// TwinCAT 3 PLC project LabExercise
// ProgramVersion: 3.1.4023.0
// libraries:
//   Tc2_NCI, * (Beckhoff Automation GmbH)
//   Tc2_Standard, * (Beckhoff Automation GmbH)
//   Tc2_System, * (Beckhoff Automation GmbH)
//   Tc3_Module, * (Beckhoff Automation GmbH)
//   VisuDialogs, * (System)
// project tree:
//   Comissioning/Function blocks/ FB_ModifyAutomaticControlSettings.TcPOU
//   Comissioning/GVLs/ G_Commissioning.TcGVL
//   Comissioning/Struct/ ST_AutomaticControlSettings.TcDUT, ST_ClosedLoopControlSettings.TcDUT, ST_MotionReferenceGeneratorSettings.TcDUT, ST_OpenLoopControlSettings.TcDUT
//   ControlBox/Interfaces/ I_ControlBox.TcIO
//   ControlBox/Function blocks/ FB_ControlBox.TcPOU, FB_RealControlBox.TcPOU, FB_VirtualControlBox.TcPOU
//   CraneControl/Function blocks/Sub blocks/ FB_ActiveDamping.TcPOU, FB_Clock.TcPOU, FB_ClosedLoopControl.TcPOU, FB_Joystick.TcPOU, FB_MotionReferenceGenerator_limit.TcPOU, FB_OpenLoopControl.TcPOU, FB_ResetIntegralController.TcPOU, FB_Status.TcPOU
//   CraneControl/Functions/ F_BarToEng.TcPOU, F_BoomAnimation.TcPOU, F_LminToEng.TcPOU, F_PistonDisplacementToBoomAngle.TcPOU, F_RadToDeg.TcPOU
//   CraneControl/Enums/ E_Mode.TcDUT, E_Status.TcDUT
//   CraneControl/Function blocks/Main blocks/ FB_AutomaticControl.TcPOU, FB_ManualControl.TcPOU
//   CraneControl/GVLs/ G_Parameters.TcGVL, G_Work.TcGVL
//   CraneControl/Struct/ ST_ActiveDamping.TcDUT, ST_AnimationScaling.TcDUT, ST_CraneKinematics.TcDUT, ST_Parameters.TcDUT, ST_RelativeMovement.TcDUT
//   / GlobalTextList.TcGTLO, PlcTask.TcTTO, Simulator.TcTTO, Visualization Manager.TcVMO (not stored)
//   HMI/ HMI.TcVIS
//   HMI/Sub/ CommissioningHMI.TcVIS, Animation.TcVIS, VirtualControlBox.TcVIS
//   ControlBox/GVLs/ G_VirtualControlBox.TcGVL
//   Programs/ MAIN.TcPOU, P_Commissioning.TcPOU, P_ControlBox.TcPOU, P_CraneControl.TcPOU, P_Simulator.TcPOU
//   Simulator/ FB_CraneSimulator.TcPOU, G_Simulator.TcGVL
// real-time tasks:
//   TASK PlcTask: cycle T#1ms, priority 20, ADS port 350
//   TASK Simulator: cycle T#100us, priority 1, ADS port 351

CONFIGURATION LabExercise
    RESOURCE PLC ON TwinCAT3
        TASK PlcTask(INTERVAL := T#1ms, PRIORITY := 20);
        TASK Simulator(INTERVAL := T#100us, PRIORITY := 1);
        PROGRAM MAIN WITH PlcTask : MAIN;
        PROGRAM P_Simulator WITH Simulator : P_Simulator;
    END_RESOURCE
END_CONFIGURATION

// ---- Comissioning/Struct/ST_AutomaticControlSettings.TcDUT
TYPE ST_AutomaticControlSettings :
STRUCT
	bEnableVelocityFeedForwardControl	: BOOL;
	bEnableClosedLoopPositionControl	: BOOL;
	bEnableIntegralController 			: BOOL;
	bEnableActiveDamping 				: BOOL;	
END_STRUCT
END_TYPE

// ---- Comissioning/Struct/ST_ClosedLoopControlSettings.TcDUT
TYPE ST_ClosedLoopControlSettings :
STRUCT
	fMaxPositionError 					: LREAL := 1E-3;
	fProportionalGain 					: LREAL := 29.17;
	fIntegralGain 						: LREAL := 19.49;
END_STRUCT
END_TYPE

// ---- Comissioning/Struct/ST_MotionReferenceGeneratorSettings.TcDUT
TYPE ST_MotionReferenceGeneratorSettings :
STRUCT
	fStartPosition_m		: LREAL := 0.0;
	fStartVelocity_m		: LREAL	:= 0.0;
	fPositionSetpoint_ms	: LREAL := 0.25;
	fVelocitySetpoint_m		: LREAL := 0.025;
	fMaxPosition 			: LREAL := 0.45;
	fMinPosition 			: LREAL := 0.0;
	fMaxVelocity 			: LREAL := 0.05;
	fTimeBeforeStarting_s	: LREAL := 3.0;
	fRampTime_s				: LREAL := 1.0;
	fHoldPositionTime_s		: LREAL := 5.0;
END_STRUCT
END_TYPE

// ---- Comissioning/Struct/ST_OpenLoopControlSettings.TcDUT
TYPE ST_OpenLoopControlSettings :
STRUCT
	fBoreArea 			: LREAL := 0.0033183;
	fAnnulusArea 		: LREAL := 0.0023562;
	fMaxFlowCapacity 	: LREAL := 30; //[l/min]
END_STRUCT
END_TYPE

// ---- CraneControl/Enums/E_Mode.TcDUT
{attribute 'qualified_only'}
{attribute 'strict'}
TYPE E_Mode :
(
	Off,
	Manual,
	Auto
);
END_TYPE

// ---- CraneControl/Enums/E_Status.TcDUT
{attribute 'qualified_only'}
{attribute 'strict'}
TYPE E_Status :
(
	Off,
	Fault,
	Ready,
	Starting,
	Running,
	Stopping,
	Checking
);
END_TYPE

// ---- CraneControl/Struct/ST_ActiveDamping.TcDUT
TYPE ST_ActiveDamping :
STRUCT
	fFlowGainInverse : LREAL := 1.7153E03;	
	fHPF_Num1 : LREAL := 9.016E-12;
	fHPF_Num2 : LREAL := -9.016E-12;
	fHPF_Den1 : LREAL := 1.0;
	fHPF_Den2 : LREAL := -0.9905;
	fVDI_Num1 : LREAL := 25;
	fVDI_Num2 : LREAL := -48.83;
	fVDI_Num3 : LREAL := 23.85;
	fVDI_Den1 : LREAL := 1;
	fVDI_Den2 : LREAL := -1.721;
	fVDI_Den3 : LREAL := 0.7408;
END_STRUCT
END_TYPE

// ---- CraneControl/Struct/ST_AnimationScaling.TcDUT
TYPE ST_AnimationScaling :
STRUCT
	fPistonScale : LREAL := 200;
	fBoomScale : LREAL := 50;
END_STRUCT
END_TYPE

// ---- CraneControl/Struct/ST_CraneKinematics.TcDUT
TYPE ST_CraneKinematics :
STRUCT
	ABx : LREAL := 0.427;
	ABy : LREAL := 1.057;
	ACx : LREAL := 0.49484;
	ACy : LREAL := 0.133;
	fBoomLength : LREAL := 3.4;
END_STRUCT
END_TYPE

// ---- CraneControl/Struct/ST_Parameters.TcDUT
TYPE ST_Parameters :
STRUCT
	fCyclicTime 						: LREAL := 0.001; //[s]
	fMaxVelocityLimit 					: LREAL := 0.05; //[m/s]
	stOpenLoopControlSettings 			: ST_OpenLoopControlSettings;
	stClosedLoopControlSettings 		: ST_ClosedLoopControlSettings;
	stPressureFeedback 					: ST_ActiveDamping;
	stCraneKinematics 					: ST_CraneKinematics;
	stAnimationScaling 					: ST_AnimationScaling;
END_STRUCT
END_TYPE

// ---- CraneControl/Struct/ST_RelativeMovement.TcDUT
TYPE ST_RelativeMovement :
STRUCT
	pt0_x : INT := 0;
	pt0_y : INT := 0;
	pt1_x : INT := 0;
	pt1_y : INT := 0; 
END_STRUCT
END_TYPE

// ---- Comissioning/GVLs/G_Commissioning.TcGVL
{attribute 'qualified_only'}
VAR_GLOBAL
	bSetNewMaxFlowCapacity		: BOOL;
	fNewMaxFlowCapacity 		: LREAL;
	bSetNewProportionalGain 	: BOOL;
	bSetNewIntegralGain 		: BOOL;
	fNewProportionalGain 		: LREAL;
	fNewIntegralGain 			: LREAL;
	bSetNewMaxPositionError 			: BOOL;
	fNewMaxPositionError				: LREAL;
	stAutomaticControlSettings 	: ST_AutomaticControlSettings;
	stMotionReferenceGeneratorSettings  : ST_MotionReferenceGeneratorSettings;
END_VAR

// ---- CraneControl/GVLs/G_Parameters.TcGVL
{attribute 'qualified_only'}
VAR_GLOBAL
	stParam : ST_Parameters;
END_VAR

// ---- CraneControl/GVLs/G_Work.TcGVL
{attribute 'qualified_only'}
VAR_GLOBAL
	eMode 			: E_Mode;
	eStatus 		: E_Status;
	fJoystickY 		: LREAL;
	bFault 			: BOOL;
	bStartButton 	: BOOL;
	bStopButton 	: BOOL;
	fControlOutputNormalized : LREAL;
END_VAR

// ---- ControlBox/GVLs/G_VirtualControlBox.TcGVL
{attribute 'qualified_only'}
VAR_GLOBAL
	bOnSelector : BOOL;
	bAutoSelector : BOOL;
	bStartButton : BOOL;
	bStopButton : BOOL;
	fJoystickY : LREAL;
	bGreenLight : BOOL;
	bRedLight : BOOL;
END_VAR

// ---- Simulator/G_Simulator.TcGVL
{attribute 'qualified_only'}
VAR_GLOBAL
	bSimulatorOn : BOOL;
	fPistonSidePressure : LREAL;
	fRodSidePressure 	: LREAL;
	fPistonPosition 	: LREAL;
	stPistonAnimation 	: ST_RelativeMovement;
	fBoomAngle 			: LREAL;
	stBoomAnimation 	: ST_RelativeMovement;
	fBoomAnimation 		: LREAL;
	fBoomAngleDeg 		: LREAL;
END_VAR

// ---- ControlBox/Interfaces/I_ControlBox.TcIO
INTERFACE I_ControlBox

METHOD Joystick
VAR_INPUT
	eMode 	: E_Mode;
	eStatus : E_Status;
END_VAR
VAR_OUTPUT
	fJoystickY : LREAL;
END_VAR
END_METHOD

METHOD Lamps 
VAR_INPUT
	eMode 	: E_Mode;
	eStatus : E_Status;
END_VAR
END_METHOD

METHOD ModeSelector 
VAR_INPUT
END_VAR
VAR_OUTPUT
	eMode : E_Mode;
END_VAR
END_METHOD

METHOD PushButtons
VAR_INPUT
	eMode 	: E_Mode;
	eStatus : E_Status;
END_VAR
VAR_OUTPUT
	bStart : BOOL;
	bStop : BOOL;
END_VAR
END_METHOD

END_INTERFACE

// ---- Programs/MAIN.TcPOU
PROGRAM MAIN
VAR
	bActivateMotion:BOOL;		//receive from ROS    sends start and stop signal
	bAuto : BOOL;				//receive from ROS    is true if we want auto mode
	bManual : BOOL;				//receive from ROS    is true if we want manual mode
	fBoomAngleRef:LREAL;			//receive from ROS	  is the desired position for the angle of the boom
	
	fPrPist : LREAL;			//sent to ROS - pressure in piston side
	fPrRod : LREAL;				//sent to ROS - pressure in rod side
	fBoomAngle:LREAL;			//sent to ROS - is the actual boom angle while crane is moving

END_VAR

P_Commissioning();
P_ControlBox();
P_CraneControl();

//SENDING TO ROS
fPrPist := G_Simulator.fPistonSidePressure;
fPrRod := G_Simulator.fRodSidePressure;
fBoomAngle := -1 * G_Simulator.fBoomAngle;


//RECEIVING FROM ROS



	
// start or stop system (through HMI buttons)
IF bActivateMotion THEN
	G_Work.bStartButton := TRUE;   //or G_Simulator.bSimulatorOn := bActivateMotion;
//ELSE
	//G_Work.bStopButton 	:= TRUE;
END_IF 

//auto or manual selection (through HMI variables)
IF bAuto THEN
	G_VirtualControlBox.bAutoSelector := FALSE;
	// set reference position
	G_VirtualControlBox.fJoystickY	:= 1 * fBoomAngleRef;				//OROR    fBoomAnimation 		: LREAL;	OR //	fBoomAngleDeg 		: LREAL;

END_IF
	
IF bManual THEN 
	G_VirtualControlBox.bAutoSelector := FALSE;
END_IF

END_PROGRAM

// ---- Programs/P_Commissioning.TcPOU
PROGRAM P_Commissioning
VAR
	fbModifyAutomaticControlSettings : FB_ModifyAutomaticControlSettings;
END_VAR

fbModifyAutomaticControlSettings(
	stParamOpenLoopControllSettings := G_Parameters.stParam.stOpenLoopControlSettings,
	bSetNewMaxFlowCapacity := G_Commissioning.bSetNewMaxFlowCapacity,
	fNewMaxFlowCapacity := G_Commissioning.fNewMaxFlowCapacity,
	stParamClosedLoopControllSettings := G_Parameters.stParam.stClosedLoopControlSettings,	
	bSetNewProportionalGain := G_Commissioning.bSetNewProportionalGain,
	fNewProportionalGain := G_Commissioning.fNewProportionalGain,
	bSetNewIntegralGain := G_Commissioning.bSetNewIntegralGain,
	fNewIntegralGain := G_Commissioning.fNewIntegralGain,
	bSetNewMaxPositionError := G_Commissioning.bSetNewMaxPositionError,
	fNewMaxPositionError := G_Commissioning.fNewMaxPositionError
);

END_PROGRAM

// ---- Comissioning/Function blocks/FB_ModifyAutomaticControlSettings.TcPOU
FUNCTION_BLOCK FB_ModifyAutomaticControlSettings
VAR_INPUT
	stParamOpenLoopControllSettings 	: REFERENCE TO ST_OpenLoopControlSettings;
	bSetNewMaxFlowCapacity				: BOOL;
	fNewMaxFlowCapacity 				: LREAL;
	stParamClosedLoopControllSettings 	: REFERENCE TO ST_ClosedLoopControlSettings;
	bSetNewProportionalGain 			: BOOL;
	bSetNewIntegralGain 				: BOOL;
	fNewProportionalGain 				: LREAL;
	fNewIntegralGain 					: LREAL;
	bSetNewMaxPositionError 			: BOOL;
	fNewMaxPositionError				: LREAL;
END_VAR
VAR_OUTPUT
END_VAR
VAR
END_VAR

IF bSetNewMaxFlowCapacity THEN
	stParamOpenLoopControllSettings.fMaxFlowCapacity := fNewMaxFlowCapacity;
	bSetNewMaxFlowCapacity := FALSE;
END_IF

IF bSetNewProportionalGain THEN
	stParamClosedLoopControllSettings.fProportionalGain := fNewProportionalGain;
	bSetNewProportionalGain := FALSE;
END_IF

IF bSetNewIntegralGain THEN
	stParamClosedLoopControllSettings.fIntegralGain := fNewIntegralGain;
	bSetNewIntegralGain := FALSE;
END_IF

IF bSetNewMaxPositionError THEN
	stParamClosedLoopControllSettings.fMaxPositionError:= fNewMaxPositionError;
	bSetNewMaxPositionError := FALSE;
END_IF

END_FUNCTION_BLOCK

// ---- Programs/P_ControlBox.TcPOU
PROGRAM P_ControlBox
VAR
	fbControlBox : FB_ControlBox; 
END_VAR

fbControlBox(
bRealControlBox := FALSE,
eStatus := G_Work.eStatus,
eMode => G_Work.eMode,
);

END_PROGRAM

// ---- ControlBox/Function blocks/FB_ControlBox.TcPOU
FUNCTION_BLOCK FB_ControlBox
VAR_INPUT
	bRealControlBox : BOOL;
	eStatus : E_Status;
END_VAR
VAR_OUTPUT
	eMode : E_Mode;
END_VAR
VAR
	fbVirtualControlBox : FB_VirtualControlBox;
	fbRealControlBox : FB_RealControlBox;
	fbSelectedControlBox : I_ControlBox := fbVirtualControlBox;
END_VAR

IF bRealControlBox THEN
	fbSelectedControlBox := fbRealControlBox;
ELSE
	fbSelectedControlBox := fbVirtualControlBox;
END_IF	
	
fbSelectedControlBox.ModeSelector(
	eMode => eMode
);

fbSelectedControlBox.PushButtons(
	eMode := eMode,
	eStatus := eStatus,
	bStart => G_Work.bStartButton,
	bStop => G_Work.bStopButton 	
);

fbSelectedControlBox.Lamps(
	eMode := eMode,
	eStatus := eStatus
);

fbSelectedControlBox.Joystick(
	eMode := eMode,
	eStatus := eStatus,
	fJoystickY => G_Work.fJoystickY
);

//IF G_Work.eStatus = E_Status.Running THEN
//	G_VirtualControlBox.bGreenLight :=  TRUE;
//ELSE
//	G_VirtualControlBox.bGreenLight :=  FALSE;
//END_IF

//IF G_Work.eStatus = E_Status.Fault THEN
//	G_VirtualControlBox.bRedLight :=  TRUE;
//ELSE
//	G_VirtualControlBox.bRedLight :=  FALSE;
//END_IF

END_FUNCTION_BLOCK

// ---- ControlBox/Function blocks/FB_VirtualControlBox.TcPOU
FUNCTION_BLOCK FB_VirtualControlBox IMPLEMENTS I_ControlBox
VAR_INPUT
END_VAR
VAR_OUTPUT
END_VAR
VAR
END_VAR

METHOD Joystick
VAR_INPUT
	eMode 	: E_Mode;
	eStatus : E_Status;
END_VAR
VAR_OUTPUT
	fJoystickY : LREAL;
END_VAR
IF eMode = E_Mode.Manual AND eStatus = E_Status.Running THEN
	fJoystickY := G_VirtualControlBox.fJoystickY;
ELSE
	fJoystickY := 0.0;
END_IF
END_METHOD

METHOD Lamps
VAR_INPUT
	eMode 	: E_Mode;
	eStatus : E_Status;
END_VAR
IF eStatus = E_Status.Running AND NOT(eMode = E_Mode.Off) THEN
	G_VirtualControlBox.bGreenLight :=  TRUE;
ELSE
	G_VirtualControlBox.bGreenLight :=  FALSE;
END_IF

IF eStatus = E_Status.Fault  AND NOT(eMode = E_Mode.Off) THEN
	G_VirtualControlBox.bRedLight :=  TRUE;
ELSE
	G_VirtualControlBox.bRedLight :=  FALSE;
END_IF
END_METHOD

METHOD ModeSelector 
VAR_INPUT
END_VAR
VAR_OUTPUT
	eMode : E_Mode;
END_VAR
CASE eMode OF 
	E_Mode.Off:	
		IF G_VirtualControlBox.bOnSelector AND NOT(G_VirtualControlBox.bAutoSelector) THEN	
			eMode := E_Mode.Manual;
		END_IF
		
		IF G_VirtualControlBox.bOnSelector AND G_VirtualControlBox.bAutoSelector THEN	
			eMode := E_Mode.Auto;
		END_IF

	E_Mode.Manual: 
		IF NOT(G_VirtualControlBox.bOnSelector) THEN	
			eMode := E_Mode.Off;
		END_IF
		
		IF G_VirtualControlBox.bOnSelector AND G_VirtualControlBox.bAutoSelector THEN	
			eMode := E_Mode.Auto;
		END_IF
	
	E_Mode.Auto:
		IF NOT(G_VirtualControlBox.bOnSelector) THEN	
			eMode := E_Mode.Off;
		END_IF
		
		IF G_VirtualControlBox.bOnSelector AND NOT(G_VirtualControlBox.bAutoSelector) THEN	
			eMode := E_Mode.Manual;
		END_IF	
ELSE 	
	eMode := E_Mode.Off;
END_CASE
END_METHOD

METHOD PushButtons
VAR_INPUT
	eMode 	: E_Mode;
	eStatus : E_Status;
END_VAR
VAR_OUTPUT
	bStart : BOOL;
	bStop : BOOL;
END_VAR
IF NOT(eMode = E_Mode.Off) AND (NOT(eStatus = E_Status.Fault) OR (eStatus = E_Status.Off)) THEN 
	bStart := G_VirtualControlBox.bStartButton;
	bStop := G_VirtualControlBox.bStopButton;
ELSE
	bStart := FALSE;
	bStop := FALSE;
END_IF
END_METHOD

END_FUNCTION_BLOCK

// ---- ControlBox/Function blocks/FB_RealControlBox.TcPOU
FUNCTION_BLOCK FB_RealControlBox IMPLEMENTS I_ControlBox
VAR_INPUT
END_VAR
VAR_OUTPUT
END_VAR
VAR
END_VAR

METHOD Joystick
VAR_INPUT
	eMode 	: E_Mode;
	eStatus : E_Status;
END_VAR
VAR_OUTPUT
	fJoystickY : LREAL;
END_VAR
END_METHOD

METHOD Lamps 
VAR_INPUT
	eMode 	: E_Mode;
	eStatus : E_Status;
END_VAR
// To Do LAB #12
END_METHOD

METHOD ModeSelector 
VAR_INPUT
END_VAR
VAR_OUTPUT
	eMode : E_Mode;
END_VAR
// To Do LAB #12
END_METHOD

METHOD PushButtons
VAR_INPUT
	eMode 	: E_Mode;
	eStatus : E_Status;
END_VAR
VAR_OUTPUT
	bStart : BOOL;
	bStop : BOOL;
END_VAR
END_METHOD

END_FUNCTION_BLOCK

// ---- Programs/P_CraneControl.TcPOU
PROGRAM P_CraneControl
VAR
 	fbStatus 					: FB_Status;
	fbRunningClock 				: FB_Clock;
	fbManualControl 			: FB_ManualControl; 
	bEnableManualControl 		: BOOL;
	fbAutomaticControl 			: FB_AutomaticControl;
	bEnableAutomaticControl 	: BOOL; 
	fbActiveDamping 			: FB_ActiveDamping;
	fControlOutputNormalized 	: LREAL; 
END_VAR

fbStatus(
bFault := G_Work.bFault,
eMode := G_Work.eMode,
fTime := fbRunningClock.fTime,
eStatus => G_Work.eStatus
);

fbRunningClock(
	bStart := (fbStatus.eStatus = E_Status.Starting) OR (fbStatus.eStatus = E_Status.Running),
	bStop := (fbStatus.eStatus = E_Status.Stopping),
	fCycleTime := G_Parameters.stParam.fCyclicTime
);

fbManualControl(
	eMode := G_Work.eMode,
	eStatus := G_Work.eStatus,
	stParam := G_Parameters.stParam, 
);

fbAutomaticControl(
	eMode := G_Work.eMode,
	eStatus := G_Work.eStatus,
	stAutomaticControlSettings := G_Commissioning.stAutomaticControlSettings,
	stMotionReferenceGeneratorSettings := G_Commissioning.stMotionReferenceGeneratorSettings,
	stParam := G_Parameters.stParam,
	fPositionFeedback := G_Simulator.fPistonPosition
);

fbActiveDamping(
	ssMethodType := BOOL_TO_SINT(G_Commissioning.stAutomaticControlSettings.bEnableActiveDamping),
	bEnable := (fbStatus.eStatus = E_Status.Running),
	stParam := G_Parameters.stParam,
	fPressurePistonSide_Pa := G_Simulator.fPistonSidePressure,
	fPressureRodSide_Pa := G_Simulator.fRodSidePressure
);
 
IF (G_Work.eMode = E_Mode.Manual AND G_Work.eStatus = E_Status.Running) THEN
	fControlOutputNormalized := LIMIT(-1.0, (fbManualControl.fControlOutputNormalized - fbActiveDamping.fPressureFeedbackNormalized), 1.0);
ELSIF (G_Work.eMode = E_Mode.Auto AND G_Work.eStatus = E_Status.Running) THEN
	fControlOutputNormalized := LIMIT(-1.0, (fbAutomaticControl.fControlOutputNormalized - fbActiveDamping.fPressureFeedbackNormalized), 1.0);
ELSE
	fControlOutputNormalized := 0.0;
END_IF

G_Work.fControlOutputNormalized := fControlOutputNormalized;

END_PROGRAM

// ---- CraneControl/Function blocks/Sub blocks/FB_Status.TcPOU
FUNCTION_BLOCK FB_Status
VAR_INPUT
	eMode 	: E_Mode;
	fTime	: LREAL;
	bFault 	: BOOL;
END_VAR
VAR_OUTPUT
	eStatus : E_Status := E_Status.Checking;
END_VAR
VAR
	bRunning : BOOL;
END_VAR

IF fTime > 2.0 THEN
	bRunning := TRUE;
ELSE
	bRunning := FALSE;	
END_IF


CASE eStatus OF 
	E_Status.Checking:
		IF bFault THEN
			eStatus := E_Status.Fault;
		END_IF
		
		IF NOT(eMode = E_Mode.Off) AND NOT(bFault)THEN	
			eStatus := E_Status.Ready;
		END_IF
		
		IF eMode = E_Mode.Off THEN	
			eStatus := E_Status.Off;
		END_IF
		
	E_Status.Off:	
		IF NOT(eMode = E_Mode.Off) THEN	
			eStatus := E_Status.Checking;
		END_IF

	E_Status.Fault:
		IF NOT(bFault) THEN
			eStatus := E_Status.Checking;
		END_IF
	
	E_Status.Ready:
		IF G_Work.bStartButton AND NOT(eMode = E_Mode.Off) AND NOT(bFault) THEN
			eStatus := E_Status.Starting;
		END_IF	
		
		IF  eMode = E_Mode.Off OR bFault THEN
			eStatus := E_Status.Checking;
		END_IF	

	E_Status.Starting:
		IF bRunning THEN
			eStatus := E_Status.Running;
		END_IF 
		
		IF bFault OR eMode = E_Mode.Off  THEN
			eStatus := E_Status.Checking;
		END_IF
		
	
	E_Status.Running:
	
		IF G_Work.bStopButton THEN
			eStatus := E_Status.Stopping;
		END_IF
		
		IF NOT(bRunning) OR eMode = E_Mode.Off OR bFault THEN
			eStatus := E_Status.Checking;
		END_IF
	
	E_Status.Stopping:	
		IF NOT(bRunning) THEN
			eStatus := E_Status.Checking;
		END_IF
	
		IF eMode = E_Mode.Off OR bFault THEN
		eStatus := E_Status.Checking;
		END_IF	
	
ELSE 	
	eStatus := E_Status.Checking;
END_CASE

END_FUNCTION_BLOCK

// ---- CraneControl/Function blocks/Sub blocks/FB_Clock.TcPOU
FUNCTION_BLOCK FB_Clock
VAR_INPUT
	bStart 		: BOOL;
	bStop 		: BOOL;
	fCycleTime  : LREAL;
END_VAR
VAR_OUTPUT
	fTime : LREAL;
END_VAR
VAR
END_VAR

IF bStart AND NOT(bStop) THEN
	fTime := fTime + fCycleTime;
ELSE
	fTime := 0.0;
END_IF

END_FUNCTION_BLOCK

// ---- CraneControl/Function blocks/Main blocks/FB_ManualControl.TcPOU
FUNCTION_BLOCK FB_ManualControl
VAR_INPUT
	eMode 	: E_Mode;
	eStatus : E_Status;
	stParam : ST_Parameters;
END_VAR
VAR_OUTPUT
	fControlOutputNormalized : LREAL;
END_VAR
VAR
	fbJoystick 			: FB_Joystick; 
	fbOpenLoopControl  	: FB_OpenLoopControl; 
END_VAR

fbJoystick(
	bEnable := (eMode = E_Mode.Manual),
	stParam := stParam,
	fNormalizedInput := G_Work.fJoystickY,
);

fbOpenLoopControl(
	bEnable := (eMode = E_Mode.Manual),
	stParam := stParam,
	fInput_ms := fbJoystick.fOuput,
	fNormalizedOutput => fControlOutputNormalized
);

END_FUNCTION_BLOCK

// ---- CraneControl/Function blocks/Sub blocks/FB_Joystick.TcPOU
FUNCTION_BLOCK FB_Joystick
VAR_INPUT
	bEnable 			: BOOL;
	fNormalizedInput 	: LREAL;
	stParam 			: ST_Parameters;
END_VAR
VAR_OUTPUT
	fOuput : LREAL;
END_VAR
VAR
END_VAR

IF bEnable THEN
	fOuput := fNormalizedInput*G_Parameters.stParam.fMaxVelocityLimit;
ELSE
	fOuput := 0.0;
END_IF

END_FUNCTION_BLOCK

// ---- CraneControl/Function blocks/Sub blocks/FB_OpenLoopControl.TcPOU
FUNCTION_BLOCK FB_OpenLoopControl
VAR_INPUT
	bEnable		: BOOL;
	fInput_ms	: LREAL;
	stParam 	: ST_Parameters;
END_VAR
VAR_OUTPUT
	fNormalizedOutput: LREAL;
END_VAR
VAR
	fFlowReference_m3s : LREAL;
	fM3sToLmin : LREAL := 60000;
END_VAR

IF fInput_ms >= 0.0 THEN 
    fFlowReference_m3s := stparam.stOpenLoopControlSettings.fBoreArea * fInput_ms;
ELSE 
    fFlowReference_m3s := fInput_ms * stparam.stOpenLoopControlSettings.fAnnulusArea;
END_IF;

IF bEnable THEN 
    fNormalizedOutput := (fM3sToLmin * fFlowReference_m3s) / stParam.stOpenLoopControlSettings.fMaxFlowCapacity;
ELSE 
    fNormalizedOutput := 0.0;
END_IF;

IF fNormalizedOutput > 1.0 THEN 
    fNormalizedOutput := 1.0;
ELSIF fNormalizedOutput < -1.0 THEN 
    fNormalizedOutput := -1.0;
END_IF;

END_FUNCTION_BLOCK

// ---- CraneControl/Function blocks/Main blocks/FB_AutomaticControl.TcPOU
FUNCTION_BLOCK FB_AutomaticControl
VAR_INPUT
	eMode 								: E_Mode;
	eStatus 							: E_Status;
	bStopMotion 						: BOOL;
	stMotionReferenceGeneratorSettings  : ST_MotionReferenceGeneratorSettings;
	stAutomaticControlSettings 			: ST_AutomaticControlSettings;
	stParam 							: ST_Parameters; 
	fPositionFeedback				 : LREAL;
END_VAR
VAR_OUTPUT
	fTime : LREAL;
	fControlOutputNormalized : LREAL;
END_VAR
VAR
	fbClock : FB_Clock;	
	fbMotionReferenceGenerator 		: FB_MotionReferenceGenerator_limit;	
	fbVelocityFeedForwardControl 	: FB_OpenLoopControl;
	fbResetIntegralController 		: FB_ResetIntegralController; 
	fbClosedLoopPositionControl 	: FB_ClosedLoopControl;
END_VAR

fbClock(
	bStart := (eMode = E_Mode.Auto AND (eStatus = E_Status.Starting OR eStatus = E_Status.Running)),
	bStop := bStopMotion,
	fCycleTime := stParam.fCyclicTime
);

fbMotionReferenceGenerator(
	bEnable := (eMode = E_Mode.Auto AND eStatus = E_Status.Running),
	stMotionReferenceGeneratorSettings := stMotionReferenceGeneratorSettings,
	fClock_s := fbClock.fTime
);

fbVelocityFeedForwardControl(
	bEnable := stAutomaticControlSettings.bEnableVelocityFeedForwardControl,
	stParam := stParam,
	fInput_ms := fbMotionReferenceGenerator.fVelocityReference_ms
);

fbResetIntegralController(
	stParam := stParam,
	fPositionError_m := fbClosedLoopPositionControl.fPositionError,
	fVelocityReference_ms := fbMotionReferenceGenerator.fVelocityReference_ms
);

fbClosedLoopPositionControl(
	bEnable := stAutomaticControlSettings.bEnableClosedLoopPositionControl,
	stParam := stParam,
	bActivateIntegralController := stAutomaticControlSettings.bEnableIntegralController,
	bIntegralControllReset := fbResetIntegralController.bReset,
	fInput_m := fbMotionReferenceGenerator.fPositionReference_m,
	fFeedback_m := fPositionFeedback
);

IF (eMode = E_Mode.Auto AND eStatus = E_Status.Running) THEN
	fControlOutputNormalized := LIMIT(-1.0, (fbVelocityFeedForwardControl.fNormalizedOutput + fbClosedLoopPositionControl.fNormalizedOutput), 1.0);
ELSE
	fControlOutputNormalized := 0.0;
END_IF

END_FUNCTION_BLOCK

// ---- CraneControl/Function blocks/Sub blocks/FB_MotionReferenceGenerator_limit.TcPOU
FUNCTION_BLOCK FB_MotionReferenceGenerator_limit
VAR_INPUT
	bEnable 							: BOOL;
	stMotionReferenceGeneratorSettings  : ST_MotionReferenceGeneratorSettings;
	fClock_s							: LREAL;
END_VAR
VAR_OUTPUT
	fPositionReference_m	: LREAL;
	fVelocityReference_ms	: LREAL;
	fTotalMotionTime_s		: LREAL;
	bErrorSignal			: BOOL;
END_VAR
VAR
	fStartPosition_m		: LREAL;
	fStartVelocity_m		: LREAL;
	fPositionSetpoint_ms	: LREAL;
	fVelocitySetpoint_m		: LREAL;
	fTimeBeforeStarting_s	: LREAL;
	fRampTime_s				: LREAL;
	fHoldPositionTime_s		: LREAL;
	Error					: DINT;
	slopeExt				: LREAL;
	slopeRetr				: LREAL;
	tHold					: LREAL;
	x1						: LREAL;
	x4						: LREAL;
	x1_tmp					: LREAL;
	x1_tmp_tmp				: LREAL;
	x4_tmp					: LREAL;
	x4_tmp_tmp				: LREAL;
	x4_tmp_tmp_0			: LREAL;
	x1_tmp_0				: LREAL;
END_VAR

IF NOT(bEnable) THEN
	RETURN;
END_IF

// LIMIT function: https://help.codesys.com/api-content/2/codesys/3.5.12.0/en/_cds_operator_limit/
fStartPosition_m := LIMIT(stMotionReferenceGeneratorSettings.fMinPosition, stMotionReferenceGeneratorSettings.fStartPosition_m, stMotionReferenceGeneratorSettings.fMaxPosition);
fStartVelocity_m := LIMIT(0.0, stMotionReferenceGeneratorSettings.fStartVelocity_m, stMotionReferenceGeneratorSettings.fMaxVelocity);
fPositionSetpoint_ms := LIMIT(stMotionReferenceGeneratorSettings.fMinPosition, stMotionReferenceGeneratorSettings.fPositionSetpoint_ms, stMotionReferenceGeneratorSettings.fMaxPosition);
fVelocitySetpoint_m := LIMIT(0.0, stMotionReferenceGeneratorSettings.fVelocitySetpoint_m, stMotionReferenceGeneratorSettings.fMaxVelocity);
fTimeBeforeStarting_s := LIMIT(0.0, stMotionReferenceGeneratorSettings.fTimeBeforeStarting_s, 10.0);
fRampTime_s := LIMIT(0.0, stMotionReferenceGeneratorSettings.fRampTime_s, 10.0);
fHoldPositionTime_s := LIMIT(0.0, stMotionReferenceGeneratorSettings.fHoldPositionTime_s, 60.0);

slopeExt := fStartVelocity_m - fVelocitySetpoint_m;

slopeRetr := ( -fVelocitySetpoint_m) - fStartVelocity_m;

tHold := ((fPositionSetpoint_ms - fStartPosition_m) - (((fVelocitySetpoint_m * fVelocitySetpoint_m) - (fStartVelocity_m * fStartVelocity_m)) / (fVelocitySetpoint_m / fRampTime_s))) / fVelocitySetpoint_m;

IF tHold < 0.0  THEN 
    bErrorSignal := TRUE;
ELSE 
    bErrorSignal := FALSE;
END_IF;

x1_tmp_tmp := fTimeBeforeStarting_s + fRampTime_s;
x1_tmp := x1_tmp_tmp - fTimeBeforeStarting_s;
x1_tmp_0 := slopeExt / fRampTime_s;
x1 := ((x1_tmp * fStartVelocity_m) + fStartPosition_m) - ((x1_tmp_0 * (x1_tmp * x1_tmp)) / 2.0);

x4_tmp_tmp := x1_tmp_tmp + tHold;
x4_tmp_tmp_0 := x4_tmp_tmp + fRampTime_s;
x4_tmp := x4_tmp_tmp_0 + fHoldPositionTime_s;
x1_tmp := x4_tmp + fRampTime_s;
x4 := x1_tmp - x4_tmp;
x4 := (fPositionSetpoint_ms - (x4 * fStartVelocity_m)) + (((slopeRetr / fRampTime_s) * (x4 * x4)) / 2.0);

IF Error = 1 THEN 
    fPositionReference_m := fStartPosition_m;
    fVelocityReference_ms := fStartVelocity_m;
ELSIF (fClock_s >= 0.0) AND (fClock_s < fTimeBeforeStarting_s) THEN 
    fPositionReference_m := fStartPosition_m;
    fVelocityReference_ms := fStartVelocity_m;
ELSIF (fClock_s >= fTimeBeforeStarting_s) AND (fClock_s < x1_tmp_tmp) THEN 
    slopeRetr := fClock_s - fTimeBeforeStarting_s;
    fPositionReference_m := ((slopeRetr * fStartVelocity_m) + fStartPosition_m) - ((x1_tmp_0 * (slopeRetr * slopeRetr)) / 2.0);
    fVelocityReference_ms := fStartVelocity_m - (x1_tmp_0 * slopeRetr);
ELSIF (fClock_s >= x1_tmp_tmp) AND (fClock_s < x4_tmp_tmp) THEN 
    fPositionReference_m := ((fClock_s - x1_tmp_tmp) * fVelocitySetpoint_m) + x1;
    fVelocityReference_ms := fVelocitySetpoint_m;
ELSIF (fClock_s >= x4_tmp_tmp) AND (fClock_s < x4_tmp_tmp_0) THEN 
    slopeRetr := fClock_s - x4_tmp_tmp;
    fPositionReference_m := ((((x4_tmp_tmp - x1_tmp_tmp) * fVelocitySetpoint_m) + x1) + (slopeRetr * fVelocitySetpoint_m)) + ((x1_tmp_0 * (slopeRetr * slopeRetr)) / 2.0);
    fVelocityReference_ms := (slopeRetr * (slopeExt / fRampTime_s)) + fVelocitySetpoint_m;
ELSIF (fClock_s >= x4_tmp_tmp_0) AND (fClock_s < x4_tmp) THEN 
    fPositionReference_m := fPositionSetpoint_ms;
    fVelocityReference_ms := fStartVelocity_m;
ELSIF (fClock_s >= x4_tmp) AND (fClock_s < x1_tmp) THEN 
    slopeExt := fClock_s - x4_tmp;
    slopeRetr := slopeRetr / fRampTime_s;
    fPositionReference_m := (fPositionSetpoint_ms - (slopeExt * fStartVelocity_m)) + ((slopeRetr * (slopeExt * slopeExt)) / 2.0);
    fVelocityReference_ms := (slopeExt * slopeRetr) + fStartVelocity_m;
ELSE 
    x1_tmp_0 := x1_tmp + tHold;

    IF (fClock_s >= x1_tmp) AND (fClock_s < x1_tmp_0) THEN 
        fPositionReference_m := x4 - ((fClock_s - x1_tmp) * fVelocitySetpoint_m);
        fVelocityReference_ms :=  -fVelocitySetpoint_m;
    ELSIF (fClock_s >= x1_tmp_0) AND (fClock_s < (((((((fTimeBeforeStarting_s + fRampTime_s) + tHold) + fRampTime_s) + fHoldPositionTime_s) + fRampTime_s) + tHold) + fRampTime_s)) THEN 
        slopeExt := fClock_s - x1_tmp_0;
        slopeRetr := slopeRetr / fRampTime_s;
        fPositionReference_m := ((x4 - ((x1_tmp_0 - x1_tmp) * fVelocitySetpoint_m)) - (slopeExt * fVelocitySetpoint_m)) - ((slopeRetr * (slopeExt * slopeExt)) / 2.0);
        fVelocityReference_ms := ( -fVelocitySetpoint_m) - (slopeExt * slopeRetr);
    ELSE 
        fPositionReference_m := fStartPosition_m;
        fVelocityReference_ms := fStartVelocity_m;
    END_IF;

END_IF;

fTotalMotionTime_s := ((((((fTimeBeforeStarting_s + fRampTime_s) + tHold) + fRampTime_s) + fHoldPositionTime_s) + fRampTime_s) + tHold) + fRampTime_s;

END_FUNCTION_BLOCK

// ---- CraneControl/Function blocks/Sub blocks/FB_ResetIntegralController.TcPOU
FUNCTION_BLOCK FB_ResetIntegralController
VAR_INPUT
	stParam 				: ST_Parameters;
	fVelocityReference_ms	: LREAL;
	fPositionError_m		: LREAL;
END_VAR
VAR_OUTPUT
	bReset: BOOL;
END_VAR
VAR
END_VAR

IF ABS(fVelocityReference_ms) > 0.0 THEN 
    bReset := FALSE;
ELSIF ABS(fPositionError_m) > stParam.stClosedLoopControlSettings.fMaxPositionError THEN 
    bReset := FALSE;
ELSE 
    bReset := TRUE;
END_IF;

END_FUNCTION_BLOCK

// ---- CraneControl/Function blocks/Sub blocks/FB_ClosedLoopControl.TcPOU
FUNCTION_BLOCK FB_ClosedLoopControl
VAR_INPUT
	bEnable						: BOOL;
	stParam 					: ST_Parameters;
	bActivateIntegralController	: BOOL;
	bIntegralControllReset		: BOOL;
	fInput_m					: LREAL;
	fFeedback_m					: LREAL;
END_VAR
VAR_OUTPUT
	fNormalizedOutput	: LREAL;
	fPositionError		: LREAL;
END_VAR
VAR
	rtb_u_FB					: LREAL;
	rtb_Saturation1				: LREAL;
	c_DiscreteTimeIntegrator_DS	: LREAL;
END_VAR

fPositionError := fInput_m - fFeedback_m;

IF bIntegralControllReset THEN 
	c_DiscreteTimeIntegrator_DS := 0.0;
END_IF;

IF c_DiscreteTimeIntegrator_DS >= 1.0 THEN 
	c_DiscreteTimeIntegrator_DS := 1.0;
ELSIF c_DiscreteTimeIntegrator_DS <= -1.0 THEN 
	c_DiscreteTimeIntegrator_DS := -1.0;
END_IF;

IF bActivateIntegralController THEN 
	rtb_u_FB := c_DiscreteTimeIntegrator_DS;
ELSE 
	rtb_u_FB := 0.0;
END_IF;

rtb_u_FB := (stParam.stClosedLoopControlSettings.fProportionalGain * fPositionError) + rtb_u_FB;

IF rtb_u_FB > 1.0 THEN 
	rtb_Saturation1 := 1.0;
ELSIF rtb_u_FB >= -1.0 THEN 
	rtb_Saturation1 := rtb_u_FB;
ELSE 
	rtb_Saturation1 := -1.0;
END_IF;

IF bEnable THEN 
	fNormalizedOutput := rtb_Saturation1;
ELSE 
	fNormalizedOutput := 0.0;
END_IF;

c_DiscreteTimeIntegrator_DS := (((((rtb_Saturation1 - rtb_u_FB) / stParam.stClosedLoopControlSettings.fProportionalGain) + fPositionError) * stParam.stClosedLoopControlSettings.fIntegralGain) * stParam.fCyclicTime) + c_DiscreteTimeIntegrator_DS;

IF c_DiscreteTimeIntegrator_DS >= 1.0 THEN 
	c_DiscreteTimeIntegrator_DS := 1.0;
ELSIF c_DiscreteTimeIntegrator_DS <= -1.0 THEN 
	c_DiscreteTimeIntegrator_DS := -1.0;
END_IF;

END_FUNCTION_BLOCK

// ---- CraneControl/Function blocks/Sub blocks/FB_ActiveDamping.TcPOU
FUNCTION_BLOCK FB_ActiveDamping
VAR_INPUT
	ssMethodType: SINT;
	bEnable: BOOL;
	stParam : ST_Parameters;
	fPressurePistonSide_Pa	: LREAL;
	fPressureRodSide_Pa		: LREAL;
END_VAR
VAR_OUTPUT
	fPressureFeedbackNormalized: LREAL;
END_VAR
VAR
	rtb_Switch3: LREAL;
	HighPassFilter_tmp: LREAL;
	VectorConcatenate: ARRAY[0..1] OF LREAL;
	VectorConcatenate1: ARRAY[0..1] OF LREAL;
	VectorConcatenate2: ARRAY[0..2] OF LREAL;
	VectorConcatenate3: ARRAY[0..2] OF LREAL;
	HighPassFilter_states: LREAL;
	ValveDynamicsInverse_states: ARRAY[0..1] OF LREAL;
END_VAR

CASE ssMethodType OF
    0: 
        HighPassFilter_states := 0.0;
        ValveDynamicsInverse_states[0] := 0.0;
        ValveDynamicsInverse_states[1] := 0.0;

    1: 
        IF bEnable THEN 
            rtb_Switch3 := 0.0;
        ELSE 
            rtb_Switch3 := 1.0;
        END_IF;

        VectorConcatenate[0] := stParam.stPressureFeedback.fHPF_Num1;
        VectorConcatenate[1] := stParam.stPressureFeedback.fHPF_Num2;
        VectorConcatenate1[0] := stParam.stPressureFeedback.fHPF_Den1;
        VectorConcatenate1[1] := stParam.stPressureFeedback.fHPF_Den2;
        VectorConcatenate2[0] := stParam.stPressureFeedback.fVDI_Num1;
        VectorConcatenate2[1] := stParam.stPressureFeedback.fVDI_Num2;
        VectorConcatenate2[2] := stParam.stPressureFeedback.fVDI_Num3;
        VectorConcatenate3[0] := stParam.stPressureFeedback.fVDI_Den1;
        VectorConcatenate3[1] := stParam.stPressureFeedback.fVDI_Den2;
        VectorConcatenate3[2] := stParam.stPressureFeedback.fVDI_Den3;

        IF rtb_Switch3 <> 0.0 THEN 
            HighPassFilter_states := 0.0;
        END_IF;

        HighPassFilter_tmp := (fPressurePistonSide_Pa - (0.7101 * fPressureRodSide_Pa)) - (VectorConcatenate1[1] * HighPassFilter_states);
		
        fPressureFeedbackNormalized := ((VectorConcatenate[0] * HighPassFilter_tmp) + (VectorConcatenate[1] * HighPassFilter_states)) * stParam.stPressureFeedback.fFlowGainInverse;

        IF fPressureFeedbackNormalized > 1.0 THEN 
            fPressureFeedbackNormalized := 1.0;
        ELSIF fPressureFeedbackNormalized < -1.0 THEN 
            fPressureFeedbackNormalized := -1.0;
        END_IF;

        IF rtb_Switch3 <> 0.0 THEN 
            ValveDynamicsInverse_states[0] := 0.0;
            ValveDynamicsInverse_states[1] := 0.0;
        END_IF;

        rtb_Switch3 := (fPressureFeedbackNormalized - (ValveDynamicsInverse_states[0] * VectorConcatenate3[1])) - (ValveDynamicsInverse_states[1] * VectorConcatenate3[2]);

        IF bEnable THEN 
            fPressureFeedbackNormalized := ((VectorConcatenate2[0] * rtb_Switch3) + (ValveDynamicsInverse_states[0] * VectorConcatenate2[1])) + (ValveDynamicsInverse_states[1] * VectorConcatenate2[2]);
        ELSE 
            fPressureFeedbackNormalized := 0.0;
        END_IF;

        IF fPressureFeedbackNormalized > 1.0 THEN 
            fPressureFeedbackNormalized := 1.0;
        ELSIF fPressureFeedbackNormalized < -1.0 THEN 
            fPressureFeedbackNormalized := -1.0;
        END_IF;

        HighPassFilter_states := HighPassFilter_tmp;

        ValveDynamicsInverse_states[1] := ValveDynamicsInverse_states[0];
        ValveDynamicsInverse_states[0] := rtb_Switch3;
END_CASE;

END_FUNCTION_BLOCK

// ---- Programs/P_Simulator.TcPOU
PROGRAM P_Simulator
VAR
	fbCraneSimulator : FB_CraneSimulator;
END_VAR

fbCraneSimulator(
	ssMethodType := BOOL_TO_SINT(G_Simulator.bSimulatorOn),
	uDCV := G_Work.fControlOutputNormalized,
	ppbar => G_Simulator.fPistonSidePressure,
	prbar => G_Simulator.fRodSidePressure,
	xm => G_Simulator.fPistonPosition
);

// Piston Animation
G_Simulator.stPistonAnimation.pt1_y := LREAL_TO_INT(fbCraneSimulator.xm * G_Parameters.stParam.stAnimationScaling.fPistonScale);
// Boom Animation
G_Simulator.fBoomAngle := F_PistonDisplacementToBoomAngle(xCyl := fbCraneSimulator.xm);
G_Simulator.fBoomAnimation := F_BoomAnimation(
	fScale := G_Parameters.stParam.stAnimationScaling.fBoomScale,
	fBoomAngle := G_Simulator.fBoomAngle,
	fBoomLength := G_Parameters.stParam.stCraneKinematics.fBoomLength,
	fBoomTipX => G_Simulator.stBoomAnimation.pt1_x,
	fBoomTipY => G_Simulator.stBoomAnimation.pt1_y
);
G_Simulator.fBoomAngleDeg := F_RadToDeg(fRad := G_Simulator.fBoomAngle);

END_PROGRAM

// ---- Simulator/FB_CraneSimulator.TcPOU
FUNCTION_BLOCK FB_CraneSimulator
VAR_INPUT
	ssMethodType: SINT;
	uDCV: LREAL;
END_VAR
VAR_OUTPUT
	xm: LREAL;
	ppbar: LREAL;
	prbar: LREAL;
END_VAR
VAR
	pLS: LREAL;
	QDCV_out: LREAL;
	rtb_xDot: LREAL;
	rtb_xDotDot: LREAL;
	temp1: LREAL;
	temp2: LREAL;
	temp3: LREAL;
	temp4: LREAL;
	c_DiscreteTimeIntegrator2_D: LREAL;
	c_DiscreteTimeIntegrator3_D: LREAL;
	c_DiscreteTimeIntegrator_DS: LREAL;
	c_DiscreteTimeIntegrator4_D: LREAL;
END_VAR



CASE ssMethodType OF
    0: 
        (* SystemInitialize for Atomic SubSystem: '<Root>/FB_CraneSimulator' *)
        (* InitializeConditions for DiscreteIntegrator: '<S1>/Discrete-Time Integrator' *)
        c_DiscreteTimeIntegrator_DS := 4.377E+6;
        (* InitializeConditions for DiscreteIntegrator: '<S1>/Discrete-Time Integrator2' *)
        c_DiscreteTimeIntegrator2_D := 0.0;
        (* InitializeConditions for DiscreteIntegrator: '<S1>/Discrete-Time Integrator3' *)
        c_DiscreteTimeIntegrator3_D := 0.0;
        (* InitializeConditions for DiscreteIntegrator: '<S1>/Discrete-Time Integrator4' *)
        c_DiscreteTimeIntegrator4_D := 468300.0;
        (* End of SystemInitialize for SubSystem: '<Root>/FB_CraneSimulator' *)
    1: 
        (* Outputs for Atomic SubSystem: '<Root>/FB_CraneSimulator' *)
        (* DiscreteIntegrator: '<S1>/Discrete-Time Integrator2' *)
        rtb_xDot := c_DiscreteTimeIntegrator2_D;
        (* Outport: '<Root>/x [m]' incorporates:
         *  DiscreteIntegrator: '<S1>/Discrete-Time Integrator3' *)
        xm := c_DiscreteTimeIntegrator3_D;
        (* Outport: '<Root>/pp [bar]' incorporates:
         *  DiscreteIntegrator: '<S1>/Discrete-Time Integrator'
         *  Gain: '<S1>/Gain' *)
        ppbar := 1.0E-5 * c_DiscreteTimeIntegrator_DS;
        (* Outport: '<Root>/pr [bar]' incorporates:
         *  DiscreteIntegrator: '<S1>/Discrete-Time Integrator4'
         *  Gain: '<S1>/Gain1' *)
        prbar := 1.0E-5 * c_DiscreteTimeIntegrator4_D;
        (* MATLAB Function: '<S1>/MATLAB Function' incorporates:
         *  DiscreteIntegrator: '<S1>/Discrete-Time Integrator'
         *  DiscreteIntegrator: '<S1>/Discrete-Time Integrator2'
         *  DiscreteIntegrator: '<S1>/Discrete-Time Integrator3'
         *  DiscreteIntegrator: '<S1>/Discrete-Time Integrator4' *)
        (* Parameters *)
        (* MATLAB Function 'FB_CraneSimulator/MATLAB Function': '<S2>:1' *)
        (* '<S2>:1:3' Fexternal = 1.3365e+04; *)
        (* [N] *)
        (* '<S2>:1:4' mEffective = 1.3365e+04; *)
        (* [kg] *)
        (* '<S2>:1:5' kFric = 4000; *)
        (* [N/(ms)] *)
        (* '<S2>:1:6' Apiston = 0.0033; *)
        (* [m^2] *)
        (* '<S2>:1:7' Aannulus = 0.0023; *)
        (* [m^2] *)
        (* '<S2>:1:8' beta = 1.0e9; *)
        (* [Pa] *)
        (* '<S2>:1:9' pSupply = 180e5; *)
        (* [Pa] *)
        (* '<S2>:1:10' pReturn = 1.1e5; *)
        (* [Pa] *)
        (* '<S2>:1:11' MaxStroke = 0.5; *)
        (* [m] *)
        (* '<S2>:1:12' VCyl_A = 1.0e-03; *)
        (* '<S2>:1:13' VCyl_B = 1.25e-03; *)
        (* '<S2>:1:14' p_nom_DCV = 7e5; *)
        (* '<S2>:1:15' Q1_ref_DCV = 20/6e4; *)
        (* '<S2>:1:16' kv1_DCV = Q1_ref_DCV/sqrt(p_nom_DCV); *)
        (* '<S2>:1:17' p0 = 7e5; *)
        (* compensator crack pressure *)
        (* Directional Control Valve - Lifting Cylinder  *)
        (* LS Pressure *)
        (* '<S2>:1:20' if uDCV > 0 *)

        IF uDCV > 0.0 THEN 
            (* '<S2>:1:21' pLS = pPiston; *)
            pLS := c_DiscreteTimeIntegrator_DS;
        ELSIF uDCV < 0.0 THEN 
            (* '<S2>:1:22' elseif uDCV < 0 *)
            (* '<S2>:1:23' pLS = pRod; *)
            pLS := c_DiscreteTimeIntegrator4_D;
        ELSE 
            (* '<S2>:1:24' else *)
            (* '<S2>:1:25' pLS = 0; *)
            pLS := 0.0;
        END_IF;

        (* '<S2>:1:28' if pLS<0 *)

        IF pLS < 0.0 THEN 
            (* '<S2>:1:29' pLS = 0; *)
            pLS := 0.0;
        END_IF;

        (* Pressure Compensator *)
        (* '<S2>:1:33' pPC = 0; *)
        (* '<S2>:1:35' if p0 <= (pSupply - pLS) *)

        IF 700000.0 <= (1.8E+7 - pLS) THEN 
            (* '<S2>:1:36' pPC = pLS+p0; *)
            pLS := pLS + 700000.0;
        ELSE 
            (* '<S2>:1:37' elseif 0 < (pSupply - pLS) < p0 *)
            (* '<S2>:1:38' pPC = pSupply-pLS; *)
            pLS := 1.8E+7 - pLS;
        END_IF;

        (* '<S2>:1:43' if pPC<0 *)

        IF pLS < 0.0 THEN 
            (* '<S2>:1:44' pPC = 0; *)
            pLS := 0.0;
        END_IF;

        (* Orifice Equations *)
        (* '<S2>:1:47' if uDCV > 0 *)

        IF uDCV > 0.0 THEN 
            (* '<S2>:1:48' QDCV_in =  kv1_DCV*uDCV*sign(pPC-pPiston)*sqrt(abs(pPC-pPiston)); *)
            pLS := pLS - c_DiscreteTimeIntegrator_DS;

            IF pLS < 0.0 THEN 
                rtb_xDotDot := -1.0;
            ELSIF pLS > 0.0 THEN 
                rtb_xDotDot := 1.0;
            ELSE 
                rtb_xDotDot := pLS;
            END_IF;

            temp3 := ABS(pLS);
            pLS := ((3.9840953644479785E-7 * uDCV) * rtb_xDotDot) * SQRT(temp3);
            (* '<S2>:1:49' QDCV_out = kv1_DCV*uDCV*sign(pRod-pReturn)*sqrt(abs(pRod-pReturn)); *)

            IF (c_DiscreteTimeIntegrator4_D - 110000.0) < 0.0 THEN 
                rtb_xDotDot := -1.0;
            ELSIF (c_DiscreteTimeIntegrator4_D - 110000.0) > 0.0 THEN 
                rtb_xDotDot := 1.0;
            ELSE 
                rtb_xDotDot := c_DiscreteTimeIntegrator4_D - 110000.0;
            END_IF;

            temp4 := ABS(c_DiscreteTimeIntegrator4_D - 110000.0);
            QDCV_out := ((3.9840953644479785E-7 * uDCV) * rtb_xDotDot) * SQRT(temp4);
        ELSIF uDCV < 0.0 THEN 
            (* '<S2>:1:50' elseif uDCV < 0 *)
            (* '<S2>:1:51' QDCV_out =  kv1_DCV*uDCV*sign(pPC-pRod)*sqrt(abs(pPC-pRod)); *)
            pLS := pLS - c_DiscreteTimeIntegrator4_D;

            IF pLS < 0.0 THEN 
                rtb_xDotDot := -1.0;
            ELSIF pLS > 0.0 THEN 
                rtb_xDotDot := 1.0;
            ELSE 
                rtb_xDotDot := pLS;
            END_IF;

            temp1 := ABS(pLS);
            QDCV_out := ((3.9840953644479785E-7 * uDCV) * rtb_xDotDot) * SQRT(temp1);
            (* '<S2>:1:52' QDCV_in =  kv1_DCV*uDCV*sign(pRod-pReturn)*sqrt(abs(pRod-pReturn)); *)

            IF (c_DiscreteTimeIntegrator4_D - 110000.0) < 0.0 THEN 
                rtb_xDotDot := -1.0;
            ELSIF (c_DiscreteTimeIntegrator4_D - 110000.0) > 0.0 THEN 
                rtb_xDotDot := 1.0;
            ELSE 
                rtb_xDotDot := c_DiscreteTimeIntegrator4_D - 110000.0;
            END_IF;

            temp2 := ABS(c_DiscreteTimeIntegrator4_D - 110000.0);
            pLS := ((3.9840953644479785E-7 * uDCV) * rtb_xDotDot) * SQRT(temp2);
        ELSE 
            (* '<S2>:1:53' else *)
            (* '<S2>:1:54' QDCV_in = 0; *)
            pLS := 0.0;
            (* '<S2>:1:55' QDCV_out = 0; *)
            QDCV_out := 0.0;
        END_IF;

        (* Pressure Gradients *)
        (* '<S2>:1:58' VA = VCyl_A + x*Apiston; *)
        (* '<S2>:1:59' VB =  VCyl_B + (MaxStroke - x)*Aannulus; *)
        (* '<S2>:1:60' VA_dot = Apiston*xDot; *)
        (* '<S2>:1:61' VB_dot = -Aannulus*xDot; *)
        (* '<S2>:1:62' pPistonDot = beta/VA*(QDCV_in - VA_dot); *)
        (* '<S2>:1:63' pRodDot = beta/VB*(-QDCV_out - VB_dot); *)
        QDCV_out := (1.0E+9 / (((0.5 - c_DiscreteTimeIntegrator3_D) * 0.0023) + 0.00125)) * (( -QDCV_out) - (-0.0023 * c_DiscreteTimeIntegrator2_D));
        (* Viscouse Friction *)
        (* '<S2>:1:66' Ffric = kFric*xDot; *)
        (* Hydraulic Force *)
        (* '<S2>:1:69' Fhyd = pPiston*Apiston - pRod*Aannulus; *)
        (* Newton Second Law of Motion *)
        (* '<S2>:1:72' xDotDot = (Fhyd - Ffric - Fexternal)/mEffective; *)
        rtb_xDotDot := ((((c_DiscreteTimeIntegrator_DS * 0.0033) - (c_DiscreteTimeIntegrator4_D * 0.0023)) - (4000.0 * c_DiscreteTimeIntegrator2_D)) - 13365.0) / 13365.0;
        (* Update for DiscreteIntegrator: '<S1>/Discrete-Time Integrator' incorporates:
         *  DiscreteIntegrator: '<S1>/Discrete-Time Integrator2'
         *  DiscreteIntegrator: '<S1>/Discrete-Time Integrator3'
         *  MATLAB Function: '<S1>/MATLAB Function' *)
        c_DiscreteTimeIntegrator_DS := (((1.0E+9 / ((c_DiscreteTimeIntegrator3_D * 0.0033) + 0.001)) * (pLS - (0.0033 * c_DiscreteTimeIntegrator2_D))) * 0.0001) + c_DiscreteTimeIntegrator_DS;

        IF c_DiscreteTimeIntegrator_DS >= 1.8E+7 THEN 
            c_DiscreteTimeIntegrator_DS := 1.8E+7;
        ELSIF c_DiscreteTimeIntegrator_DS <= 110000.0 THEN 
            c_DiscreteTimeIntegrator_DS := 110000.0;
        END_IF;

        (* End of Update for DiscreteIntegrator: '<S1>/Discrete-Time Integrator' *)
        

        (* Update for DiscreteIntegrator: '<S1>/Discrete-Time Integrator2' *)
        c_DiscreteTimeIntegrator2_D := (0.0001 * rtb_xDotDot) + c_DiscreteTimeIntegrator2_D;

        IF c_DiscreteTimeIntegrator2_D >= 0.12 THEN 
            c_DiscreteTimeIntegrator2_D := 0.12;
        ELSIF c_DiscreteTimeIntegrator2_D <= -0.12 THEN 
            c_DiscreteTimeIntegrator2_D := -0.12;
        END_IF;

        (* End of Update for DiscreteIntegrator: '<S1>/Discrete-Time Integrator2' *)
        

        (* Update for DiscreteIntegrator: '<S1>/Discrete-Time Integrator3' *)
        c_DiscreteTimeIntegrator3_D := (0.0001 * rtb_xDot) + c_DiscreteTimeIntegrator3_D;

        IF c_DiscreteTimeIntegrator3_D >= 0.5 THEN 
            c_DiscreteTimeIntegrator3_D := 0.5;
        ELSIF c_DiscreteTimeIntegrator3_D <= 0.0 THEN 
            c_DiscreteTimeIntegrator3_D := 0.0;
        END_IF;

        (* End of Update for DiscreteIntegrator: '<S1>/Discrete-Time Integrator3' *)
        

        (* Update for DiscreteIntegrator: '<S1>/Discrete-Time Integrator4' *)
        c_DiscreteTimeIntegrator4_D := (0.0001 * QDCV_out) + c_DiscreteTimeIntegrator4_D;

        IF c_DiscreteTimeIntegrator4_D >= 1.8E+7 THEN 
            c_DiscreteTimeIntegrator4_D := 1.8E+7;
        ELSIF c_DiscreteTimeIntegrator4_D <= 110000.0 THEN 
            c_DiscreteTimeIntegrator4_D := 110000.0;
        END_IF;

        (* End of Update for DiscreteIntegrator: '<S1>/Discrete-Time Integrator4' *)
        (* End of Outputs for SubSystem: '<Root>/FB_CraneSimulator' *)
END_CASE;

END_FUNCTION_BLOCK

// ---- CraneControl/Functions/F_PistonDisplacementToBoomAngle.TcPOU
FUNCTION F_PistonDisplacementToBoomAngle : LREAL
VAR_INPUT
	xCyl : LREAL;
END_VAR
VAR
	AB : LREAL;
	AC : LREAL;
	BC : LREAL;
	alpha1 : LREAL;
	alpha2 : LREAL;
	theta1 : LREAL;
	AB2 : LREAL;
	AC2 : LREAL;
	BC2 : LREAL;
END_VAR

AB := SQRT(ABS(G_Parameters.stParam.stCraneKinematics.ABx)*ABS(G_Parameters.stParam.stCraneKinematics.ABx) + ABS(G_Parameters.stParam.stCraneKinematics.ABy)*ABS(G_Parameters.stParam.stCraneKinematics.ABy));
AC := SQRT(ABS(G_Parameters.stParam.stCraneKinematics.ACx)*ABS(G_Parameters.stParam.stCraneKinematics.ACx) + ABS(G_Parameters.stParam.stCraneKinematics.ACy)*ABS(G_Parameters.stParam.stCraneKinematics.ACy));

BC := 0.77222 + xCyl;

alpha1 := ATAN(ABS(G_Parameters.stParam.stCraneKinematics.ACy)/ ABS(G_Parameters.stParam.stCraneKinematics.ACx));
alpha2 := ATAN(ABS(G_Parameters.stParam.stCraneKinematics.ABy)/ ABS(G_Parameters.stParam.stCraneKinematics.ABx));

AB2 := ABS(AB)*ABS(AB);
AC2 := ABS(AC)*ABS(AC);
BC2 := ABS(BC)*ABS(BC);

theta1 := ACOS( (AB2 + AC2 - BC2) / (2 * ABS(AB) * ABS(AC)) ) - alpha2 + alpha1;

F_PistonDisplacementToBoomAngle := theta1;

END_FUNCTION

// ---- CraneControl/Functions/F_BoomAnimation.TcPOU
FUNCTION F_BoomAnimation 
VAR_INPUT
	fScale : LREAL;
	fBoomAngle : LREAL;
	fBoomLength : LREAL;
END_VAR
VAR_OUTPUT
	fBoomTipX : INT;
	fBoomTipY : INT;
END_VAR
VAR
END_VAR

fBoomTipX := LREAL_TO_INT( fBoomLength * ( COS(fBoomAngle) - SIN(fBoomAngle) ) * fScale );
fBoomTipY := LREAL_TO_INT( fBoomLength * ( SIN(fBoomAngle) + COS(fBoomAngle) ) * fScale );

END_FUNCTION

// ---- CraneControl/Functions/F_RadToDeg.TcPOU
FUNCTION F_RadToDeg : LREAL
VAR_INPUT
	fRad : LREAL;
END_VAR
VAR
END_VAR

F_RadToDeg := fRad * (180/PI);

END_FUNCTION

// ---- CraneControl/Functions/F_BarToEng.TcPOU
FUNCTION F_BarToEng : LREAL
VAR_INPUT
	fBar : LREAL;
END_VAR
VAR
END_VAR

F_BarToEng := fBar*1E5;

END_FUNCTION

// ---- CraneControl/Functions/F_LminToEng.TcPOU
FUNCTION F_LminToEng : LREAL
VAR_INPUT
	fLmin : LREAL;
END_VAR
VAR
END_VAR

F_LminToEng := fLmin / 60000;

END_FUNCTION

// ---- GlobalTextList.TcGTLO
TEXTLIST GlobalTextList
  624 = '%0.1f'
  198 = '%f'
  949 = '%i'
  819 = '%s'
  850 = '%s '
  935 = '0.5m'
  892 = '0m'
  807 = '1m'
  948 = '1mx0'
  858 = 'Active Damping ON'
  91 = 'Animation'
  175 = 'AUTO'
  885 = 'Automatic Control Settings'
  104 = 'Boom Angle: %0.1f [deg]'
  236 = 'Clock: %s [s]'
  920 = 'Closed Loop Position Control ON'
  214 = 'Comissioning'
  52 = 'ControlBox'
  109 = 'Controller Parameter Tuning'
  829 = 'Current I-gain: %0.1f '
  58 = 'Current Max Piston Stroke: %0.1f [m] '
  577 = 'Current MaxError: %0.1f '
  147 = 'Current MaxError: %0.1f [m] '
  196 = 'Current MaxError: %f [m] '
  955 = 'Current MaxFlow: %0.1f [L/min] '
  827 = 'Current MaxFlow: %0.1f [m] '
  137 = 'Current P-gain: %0.1f '
  668 = 'Current P-gain: %0.1f [m] '
  791 = 'Current Pgain: %0.1f [m] '
  471 = 'Cylinder Position Reference: %0.1f [m]'
  995 = 'Cylinder Position Reference: %f [m]'
  752 = 'Cylinder Velocity Reference: %0.0001f [m/s]'
  954 = 'Cylinder Velocity Reference: %0.01f [m/s]'
  105 = 'Cylinder Velocity Reference: %0.1f [m/s]'
  755 = 'Cylinder Velocity Reference: %0.1s [m/s]'
  25 = 'Cylinder Velocity Reference: %f [m/s]'
  308 = 'Cylinder Velocity Reference: %f [m]'
  30 = 'Cylinder Velocity Reference: %i'
  903 = 'Cylinder Velocity Reference: %s'
  128 = 'Cylinder Velocity Reference: %s [m/s]'
  353 = 'Enable'
  409 = 'ENABLE'
  527 = 'End Stop Status: %s '
  90 = 'FAULT'
  548 = 'Feed Forward Controller On'
  392 = 'Feed Forward Tuning'
  187 = 'Gain'
  904 = 'Hold Pos time: %0.1f [s] '
  445 = 'Integral Controller'
  81 = 'Integral Controller Gain'
  443 = 'Integral Controller On'
  573 = 'Integral Controller ON'
  961 = 'JOYSTICK Y'
  660 = 'MANUAL'
  8 = 'Manual Cylinder Position   Reference [m]'
  157 = 'Manual Cylinder Position Reference'
  11 = 'Manual Cylinder Position Reference [m]'
  7 = 'Max Piston Stroke: %0.1f [m] '
  110 = 'Max Piston Stroke: %f [m] '
  261 = 'Max Position Error'
  84 = 'Max Stroke: %f [m] '
  188 = 'Mode'
  76 = 'Mode: %s '
  415 = 'Motion Reference Generator Settings'
  655 = 'New I-gain: %0.1f '
  646 = 'New Max Piston Stroke: %0.1f [m] '
  895 = 'New MaxError: %0.1f '
  731 = 'New MaxError: %0.1f  [m]'
  683 = 'New MaxError: %f  [m]'
  330 = 'New MaxFlow: %0.1f [L/min] '
  993 = 'New MaxFlow: %0.1f [m] '
  347 = 'New P-gain: %0.1f '
  792 = 'New P-gain: %0.1f [m] '
  65 = 'OFF'
  629 = 'ON'
  751 = 'Pgain: %0.1f [m] '
  622 = 'Position SP: %0.1f [m] '
  463 = 'Position SP: %f [m] '
  651 = 'Proportional '
  705 = 'Proportional  Controller'
  982 = 'Proportional  Controller Gain'
  711 = 'Proportional Gain'
  215 = 'Ramp time: %0.1f [s] '
  310 = 'RUNNING'
  695 = 'Set New Value'
  466 = 'Simulation'
  9 = 'Simulator ON'
  279 = 'Start'
  868 = 'START'
  254 = 'START AUTO'
  149 = 'Start delay: %0.1f [m/s] '
  828 = 'Start delay: %0.1f [s] '
  324 = 'Start Position SP: %0.1f [m/s] '
  286 = 'Start Position: %0.1f [m] '
  78 = 'Start Position: %f [m] '
  253 = 'Start Velocity %0.1f [m/s] '
  314 = 'Start Velocity: %0.1f [m/s] '
  983 = 'Start Velocity: %f [m/s] '
  978 = 'Started'
  795 = 'Status'
  173 = 'Status: %s '
  397 = 'STOP'
  495 = 'Time: %0.1f [s]'
  221 = 'Time: %f [s]'
  61 = 'Time: %i [s]'
  725 = 'Time: %s [s]'
  638 = 'Velocity SP: %0.1f [m/s] '
  999 = 'Velocity SP: %f [m/s] '
  730 = 'VelocityFeed Forward Controller On'
  560 = 'VelocityFeed Forward Controller ON'
  444 = 'x0'
END_TEXTLIST

// ---- HMI/HMI.TcVIS
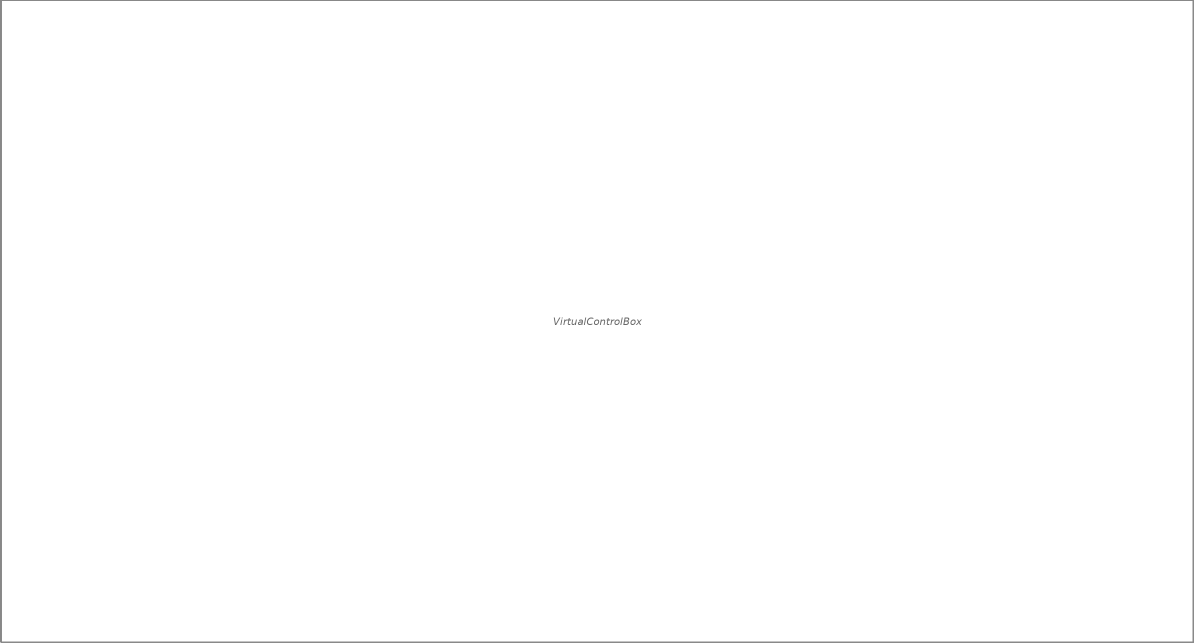
VISUALIZATION HMI  // 1194x643
    TabControl (1,0 1193x643)
        shows VirtualControlBox()
        shows CommissioningHMI()
        shows Animation()
        [0]: TabTitle=ControlBox
        [1]: TabTitle=Comissioning
        [2]: TabTitle=Animation
END_VISUALIZATION

// ---- HMI/Sub/CommissioningHMI.TcVIS
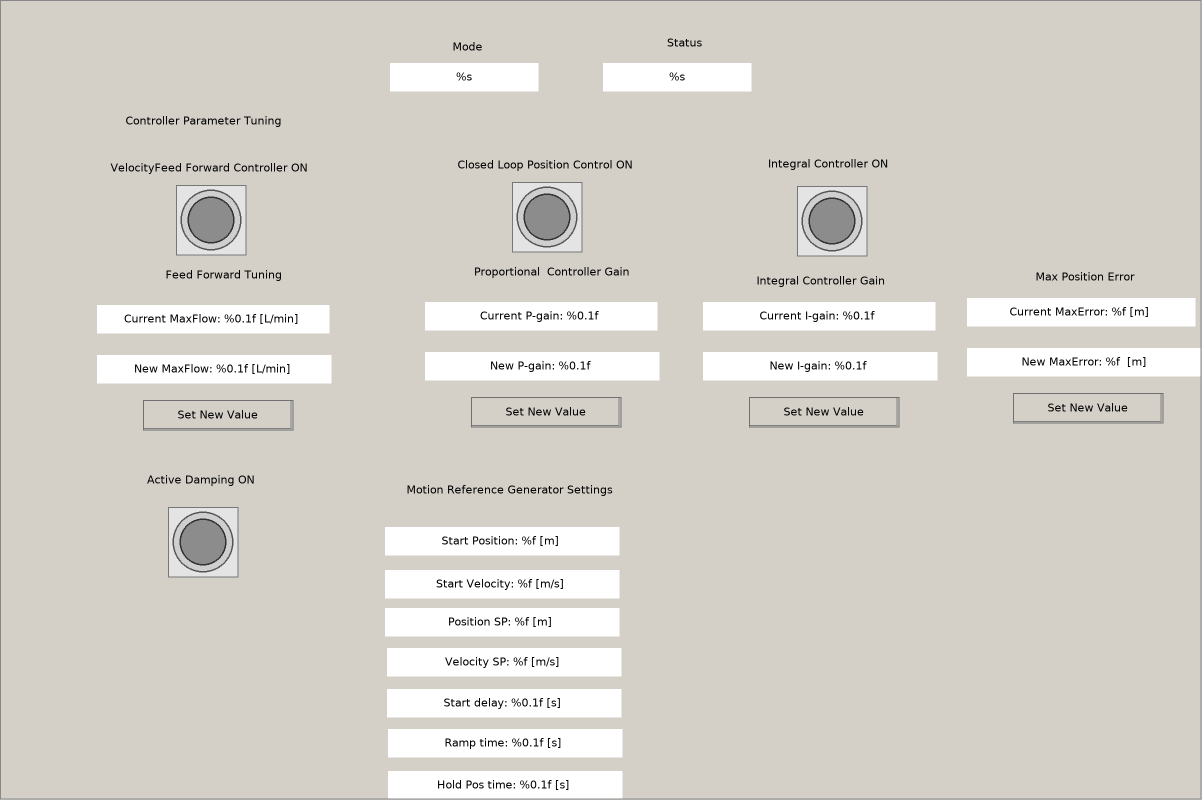
VISUALIZATION CommissioningHMI  // 1202x800
    Button (471,397 150x30), "Set New Value"
        tap G_Commissioning.bSetNewProportionalGain
    Textfield (424,301 234x30), "Current P-gain: %0.1f", text variable: G_Parameters.stParam.stClosedLoopControlSettings.fProportionalGain
    Textfield (424,351 236x30), "New P-gain: %0.1f", text variable: G_Commissioning.fNewProportionalGain
        OnMouseDown: write the text variable via Default
    Label (469,257 166x30), "Proportional Controller Gain"
    Button (749,397 150x30), "Set New Value"
        tap G_Commissioning.bSetNewIntegralGain
    Textfield (702,301 234x30), "Current I-gain: %0.1f", text variable: G_Parameters.stParam.stClosedLoopControlSettings.fIntegralGain
    Textfield (702,351 236x30), "New I-gain: %0.1f", text variable: G_Commissioning.fNewIntegralGain
        OnMouseDown: write the text variable via Default
    Label (746,266 150x30), "Integral Controller Gain"
    Label (94,106 219x30), "Controller Parameter Tuning"
    PushSwitch (797,186 70x70), variable: G_Commissioning.stAutomaticControlSettings.bEnableIntegralController, behaviour: TOGGLE, style: Switch-PushSwitch-Gray
    Label (745,149 166x30), "Integral Controller ON"
    Label (419,150 252x30), "Closed Loop Position Control ON"
    PushSwitch (512,182 70x70), variable: G_Commissioning.stAutomaticControlSettings.bEnableClosedLoopPositionControl, behaviour: TOGGLE, style: Switch-PushSwitch-Gray
    Label (83,153 252x30), "VelocityFeed Forward Controller ON"
    PushSwitch (176,185 70x70), variable: G_Commissioning.stAutomaticControlSettings.bEnableVelocityFeedForwardControl, behaviour: TOGGLE, style: Switch-PushSwitch-Gray
    PushSwitch (168,507 70x70), variable: G_Commissioning.stAutomaticControlSettings.bEnableActiveDamping, behaviour: TOGGLE, style: Switch-PushSwitch-Gray
    Label (75,465 252x30), "Active Damping ON"
    Button (143,400 150x30), "Set New Value"
        tap G_Commissioning.bSetNewMaxFlowCapacity
    Textfield (96,304 234x30), "Current MaxFlow: %0.1f [L/min]", text variable: G_Parameters.stParam.stOpenLoopControlSettings.fMaxFlowCapacity
    Textfield (96,354 236x30), "New MaxFlow: %0.1f [L/min]", text variable: G_Commissioning.fNewMaxFlowCapacity
        OnMouseDown: write the text variable via Default, min 0, max 40
    Label (141,260 166x30), "Feed Forward Tuning"
    Button (1013,393 150x30), "Set New Value"
        tap G_Commissioning.bSetNewMaxPositionError
    Textfield (966,297 230x30), "Current MaxError: %f [m]", text variable: G_Parameters.stParam.stClosedLoopControlSettings.fMaxPositionError
    Textfield (966,347 236x30), "New MaxError: %f [m]", text variable: G_Commissioning.fNewMaxPositionError
        OnMouseDown: write the text variable via Default
    Label (1010,262 150x30), "Max Position Error"
    Label (412,32 111x30), "Mode"
    Label (629,28 111x30), "Status"
    Textfield (389,62 150x30), "%s", text variable: G_Work.eMode
    Textfield (602,62 150x30), "%s", text variable: G_Work.eStatus
    Label (364,475 291x30), "Motion Reference Generator Settings"
    Textfield (384,526 236x30), "Start Position: %f [m]", text variable: G_Commissioning.stMotionReferenceGeneratorSettings.fStartPosition_m
        OnMouseDown: write the text variable via Default, min 0, max 0.5
    Textfield (384,569 236x30), "Start Velocity: %f [m/s]", text variable: G_Commissioning.stMotionReferenceGeneratorSettings.fStartVelocity_m
        OnMouseDown: write the text variable via Default, min 0, max 0.05
    Textfield (384,607 236x30), "Position SP: %f [m]", text variable: G_Commissioning.stMotionReferenceGeneratorSettings.fPositionSetpoint_ms
        OnMouseDown: write the text variable via Default, min 0, max 0.45
    Textfield (386,647 236x30), "Velocity SP: %f [m/s]", text variable: G_Commissioning.stMotionReferenceGeneratorSettings.fVelocitySetpoint_m
        OnMouseDown: write the text variable via Default, min 0, max 0.05
    Textfield (386,688 236x30), "Start delay: %0.1f [s]", text variable: G_Commissioning.stMotionReferenceGeneratorSettings.fTimeBeforeStarting_s
        OnMouseDown: write the text variable via Default, min 0, max 10
    Textfield (387,728 236x30), "Ramp time: %0.1f [s]", text variable: G_Commissioning.stMotionReferenceGeneratorSettings.fRampTime_s
        OnMouseDown: write the text variable via Default, min 0, max 10
    Textfield (387,770 236x30), "Hold Pos time: %0.1f [s]", text variable: G_Commissioning.stMotionReferenceGeneratorSettings.fHoldPositionTime_s
        OnMouseDown: write the text variable via Default, min 0, max 10
END_VISUALIZATION

// ---- HMI/Sub/Animation.TcVIS
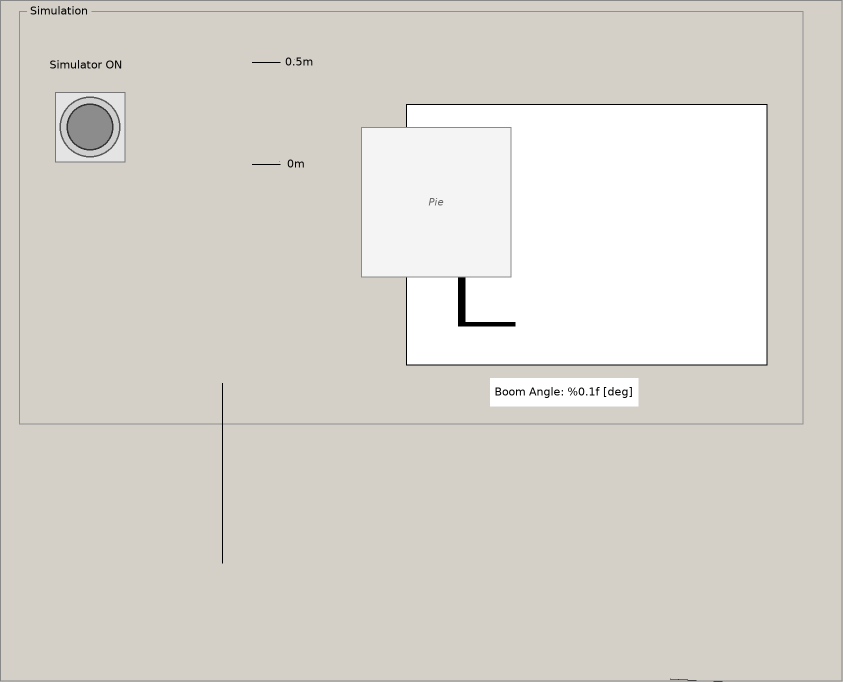
VISUALIZATION Animation  // 843x682
    GroupBox (19,3 784x421), "Simulation"
        Rectangle (387,101 361x261)
        Line (233,161) (261,161)
        Label (263,146 28x30), "0m"
        Line (233,59) (261,59)
        Textfield (470,374 150x30), "Boom Angle: %0.1f [deg]", text variable: G_Simulator.fBoomAngleDeg
        Rectangle (439,265 7x58)
        Rectangle (440,319 56x4)
        PushSwitch (36,89 70x70), variable: G_Simulator.bSimulatorOn, behaviour: TOGGLE, style: Switch-PushSwitch-Gray
    Line (222,383) (222,563)
        p1126004900: G_Simulator.stPistonAnimation.pt1_y
        p3528305787: G_Simulator.stPistonAnimation.pt0_x
        p2773130477: G_Simulator.stPistonAnimation.pt0_y
        p874137650: G_Simulator.stPistonAnimation.pt1_x
    Line (279,161) (279,161)
    Label (285,47 28x30), "0.5m"
    Line (294,59) (294,59)
    Line (722,682) (670,679)
        p1126004900: G_Simulator.stBoomAnimation.pt1_y
        p3528305787: G_Simulator.stBoomAnimation.pt0_x
        p2773130477: G_Simulator.stBoomAnimation.pt0_y
        p874137650: -G_Simulator.stBoomAnimation.pt1_x
    Label (-40,50 252x30), "Simulator ON"
    Pie (361,127 150x150)
END_VISUALIZATION

// ---- HMI/Sub/VirtualControlBox.TcVIS
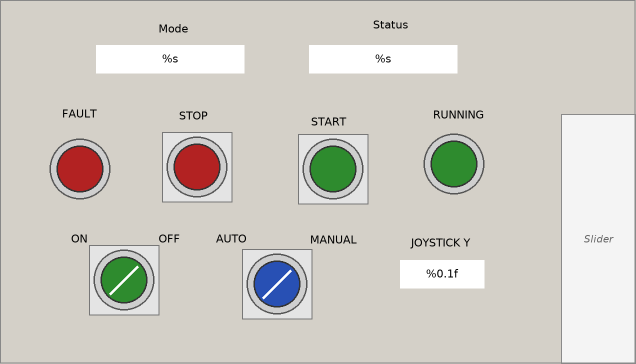
VISUALIZATION VirtualControlBox  // 636x364
    Lamp1 (419,129 70x70), variable: G_VirtualControlBox.bGreenLight, style: Lamp-Lamp1-Green
    Lamp1 (45,134 70x70), variable: G_VirtualControlBox.bRedLight, style: Lamp-Lamp1-Red
    PushSwitch (162,132 70x70), variable: G_VirtualControlBox.bStopButton, behaviour: TAP, style: Switch-PushSwitch-Red
    PushSwitch (298,134 70x70), variable: G_VirtualControlBox.bStartButton, behaviour: TAP, style: Switch-PushSwitch-Green
    RotarySwitch (89,245 70x70), variable: G_VirtualControlBox.bOnSelector, behaviour: TOGGLE, style: Switch-RotarySwitch-Green
    Label (51,224 57x30), "ON"
    Label (141,224 57x30), "OFF"
    RotarySwitch (242,249 70x70), variable: G_VirtualControlBox.bAutoSelector, behaviour: TOGGLE, style: Switch-RotarySwitch-Blue
    Label (203,224 57x30), "AUTO"
    Label (305,225 57x30), "MANUAL"
    Slider (561,114 75x250), variable: G_VirtualControlBox.fJoystickY, scale -1..1
    Label (51,99 57x30), "FAULT"
    Label (430,100 57x30), "RUNNING"
    Label (300,107 57x30), "START"
    Label (165,101 57x30), "STOP"
    Label (385,228 111x30), "JOYSTICK Y"
    Textfield (399,259 86x30), "%0.1f", text variable: G_VirtualControlBox.fJoystickY
        OnMouseClick: write the text variable via Default, min -1, max 1
    Label (118,14 111x30), "Mode"
    Label (335,10 111x30), "Status"
    Textfield (95,44 150x30), "%s", text variable: G_Work.eMode
    Textfield (308,44 150x30), "%s", text variable: G_Work.eStatus
END_VISUALIZATION
